// TIA Portal project "XC221_TRABALHOSO" (V12)

(* hardware
DEVICE "S7-1200 station_1"  SIMATIC 1200-Station
   slot 0: "S7-1200 rack"  Rack  V1.0
   slot 1: "PLC_123"  CPU 1214C DC/DC/DC  6ES7 214-1AG31-0XB0  V3.0
   slot 3: "AQ1 x 12 bits"  6ES7 232-4HA30-0XB0  V1.0
*)

// ===== PLC "PLC_123"  CPU 1214C DC/DC/DC =====
// protected blocks, not shown: "EASYPI", "MEMRST"

VAR_GLOBAL   // PLC tag table "Default tag table"
   "System_Byte" AT %MB1 : Byte;
   "FirstScan" AT %M1.0 : Bool;
   "DiagStatusUpdate" AT %M1.1 : Bool;
   "AlwaysTRUE" AT %M1.2 : Bool;
   "AlwaysFALSE" AT %M1.3 : Bool;
   "Clock_Byte" AT %MB0 : Byte;
   "Clock_10Hz" AT %M0.0 : Bool;
   "Clock_5Hz" AT %M0.1 : Bool;
   "Clock_2.5Hz" AT %M0.2 : Bool;
   "Clock_2Hz" AT %M0.3 : Bool;
   "Clock_1.25Hz" AT %M0.4 : Bool;
   "Clock_1Hz" AT %M0.5 : Bool;
   "Clock_0.625Hz" AT %M0.6 : Bool;
   "Clock_0.5Hz" AT %M0.7 : Bool;
   "Tag_1" AT %M31.0 : Bool;
   "Comando_ventilador1" AT %M31.1 : Bool;   // Variavel Auxliar usado no Ventilado 1
   "Comando_ventilador2" AT %M31.2 : Bool;   // Variavel Auxliar usado no Ventilado 2
   "Tag_2" AT %MD701 : Real;
   "Tag_3" AT %MD573 : Real;
   "Tag_4" AT %M203.2 : Bool;
   "Comando_ventilador3" AT %M203.3 : Bool;   // Variavel Auxliar usado no Ventilado 3
   "Comando_ventilador4" AT %M203.4 : Bool;   // Variavel Auxliar usado no Ventilado 4
END_VAR

VAR_GLOBAL   // PLC tag table "11 - Parâmetros"
   "Par_VT101_HorLim" AT %MD705 : Real;   // Limite de Horas do Ventilador 1
   "Par_VT102_HorLim" AT %MD709 : Real;   // Limite de Horas do Ventilador 2
   "Par_LT101_LimHH" AT %MD713 : Real;   // Limite para a condição “Muito Alto” [mm]
   "Par_LT101_LimH" AT %MD717 : Real;   // Limite para a condição “Alto” [mm]
   "Par_LT101_LimL" AT %MD721 : Real;   // Limite para a condição “Baixo" [mm]
   "Par_LT101_LimLL" AT %MD725 : Real;   // Limite para a condição “Muito Baixo” [mm]
   "Par_LT101_LimDsg" AT %MD729 : Real;   // Limite para desligar a bomba[mm]
   "Par_LT101_LimLig" AT %MD733 : Real;   // Limite para ligar a bomba [mm]
   "Par_LC102_SetPoint" AT %MD737 : Real;   // Setpoint [mm]
   "Par_LC102_Prop" AT %MD741 : Real;   // Ganho proporcional
   "Par_LC102_Integ" AT %MD745 : Real;   // Ganho integral [segundos]
   "Par_BA101_HorLim" AT %MD753 : Real;   // Limite de horas da bomba
   "Par_BA101_RefVel" AT %MD757 : Real;   // Referência de velocidade da bomba [%]
END_VAR

VAR_GLOBAL   // PLC tag table "01 - Entradas Digitais"
   "DIn_Geral_Emerge" AT %I0.0 : Bool;   // Ativa condição de emergencia
   "DIn_Geral_Rearma" AT %I0.1 : Bool;   // Rearma defeitos
   "DIn_Geral_SelLoc" AT %I0.2 : Bool;   // Seleciona local (valvula e ventiladores)
   "DIn_VS101_Abre" AT %I0.3 : Bool;   // Botão abre valvula
   "DIn_VS101_Fecha" AT %I0.4 : Bool;   // Botao fecha valvula
   "DIn_VT101_LigDsg" AT %I0.5 : Bool;   // Botão liga/desliga ventilador 1
   "DIn_VT102_LigDsl" AT %I0.6 : Bool;   // Botão liga/desliga ventilador 2
   "DIn_BA101_DisjOff" AT %I0.7 : Bool;   // Disjuntor da bomba desarmado
END_VAR

VAR_GLOBAL   // PLC tag table "02 - Saidas Digitais"
   "Dou_VS101_Abre" AT %Q0.0 : Bool;   // Abre valvula (energiza)
   "Dou_VT101_Liga" AT %Q0.1 : Bool;   // Liga ventilador 1 (energiza)
   "DOu_VT102_Liga" AT %Q0.2 : Bool;   // Liga ventilador 2 (energiza)
END_VAR

VAR_GLOBAL   // PLC tag table "03 - Entradas Analogicas"
   "AIn_LT101_Nivel" AT %IW64 : UInt;   // Nivel de água no tanque [bruto]
END_VAR

VAR_GLOBAL   // PLC tag table "04 - Saidas Analogicas"
   "AOu_BA101_VelBmb" AT %QW64 : UInt;   // Velocidade da bomba [bruto]
END_VAR

VAR_GLOBAL   // PLC tag table "05 - Comando"
   "Cmd_GERAL_Rearma" AT %M101.0 : Bool;   // Rearma defeitos
   "Cmd_VS101_Abre" AT %M102.0 : Bool;   // Abre valvula
   "Cmd_VS101_Fecha" AT %M102.1 : Bool;   // Fecha valvula
   "Cmd_VT101_Liga" AT %M103.0 : Bool;   // Liga ventilador 1
   "Cmd_VT101_Deslig" AT %M103.1 : Bool;   // Desliga ventilador 1
   "Cmd_VT101_HorRst" AT %M103.2 : Bool;   // Zera horimetro ventilador 1
   "Cmd_VT102_Liga" AT %M104.0 : Bool;   // Liga ventilador 2
   "Cmd_VT102_Deslig" AT %M104.1 : Bool;   // Desliga ventilador 2
   "Cmd_VT102_HorRst" AT %M104.2 : Bool;   // Zera horimetro do ventilador 2
   "Cmd_BA101_Liga" AT %M108.0 : Bool;   // Liga bomba
   "Cmd_BA101_Deslig" AT %M108.1 : Bool;   // Desliga bomba
   "Cmd_BA101_HorRst" AT %M108.2 : Bool;   // Zera horimetro da bomba
   "Cmd_BA101_SelMan" AT %M108.3 : Bool;   // Seleciona modo manual da bomba
   "Cmd_BA101_SelAut" AT %M108.4 : Bool;   // Seleciona modo automatico da bomba
   "Cmd_BA101_SelPID" AT %M108.5 : Bool;   // Seleciona modo PID da bomba
   "Cmd_BA101_SelOnOff" AT %M108.6 : Bool;   // Seleciona modo On/Off da bomba
END_VAR

VAR_GLOBAL   // PLC tag table "06 - Estados"
   "STT_geral_LocSel" AT %M201.0 : Bool;   // Local selecionado(Válvula e ventiladores)
   "STT_VS101_Aberta" AT %M202.0 : Bool;   // Válvula aberta(energizada)
   "STT_VT101_Ligado" AT %M203.0 : Bool;   // Ventilador 1 ligado
   "STT_VT101_Defeito" AT %M203.1 : Bool;   // Ventilador 1 com defeito
   "STT_VT102_Ligado" AT %M204.0 : Bool;   // Ventilador 2 ligado
   "STT_VT102_Defeito" AT %M204.1 : Bool;   // Ventilador 2 com defeito
   "STT_LC101_LigBmb" AT %M206.0 : Bool;   // Solicitação do controlador ON/OFF para ligar a bomba
   "STT_BA101_Ligada" AT %M208.0 : Bool;   // Bomba ligada
   "STT_BA101_Defeito" AT %M208.1 : Bool;   // Bomba com defeito
   "STT_BA101_Bloq" AT %M208.2 : Bool;   // Bomba bloqueada
   "STT_BA101_Mansel" AT %M208.3 : Bool;   // Bomba em modo manual
   "STT_BA101_PIDsel" AT %M208.4 : Bool;   // Bomba em modo PID
END_VAR

VAR_GLOBAL   // PLC tag table "07 - Alarmes"
   "Alr_Geral_emerge" AT %M301.0 : Bool;   // Condição de emergencia ativada
   "Alr_VT101_Horfim" AT %M303.0 : Bool;   // Ventilador 1 com horas esgotadas
   "Alr_VT102_Horfim" AT %M304.0 : Bool;   // Ventilador 2 com horas esgotadas
   "Alr_LT101_ExcedHH" AT %M305.0 : Bool;   // Limite "Muito alto" excedido
   "Alr_LT101_ExcedH" AT %M305.1 : Bool;   // limite "alto" excedido
   "Alr_LT101_ExcedL" AT %M305.2 : Bool;   // limite "baixo" excedido
   "Alr_LT101_ExcedLL" AT %M305.3 : Bool;   // limite "muito baixo" excedido
   "Alr_BA101_HorFim" AT %M308.0 : Bool;   // Bomba com horas esgotadas
   "Alr_BA101_DisjOff" AT %M308.1 : Bool;   // Disjuntor da bomba desarmado
END_VAR

VAR_GLOBAL   // PLC tag table "08 - Auxiliares Digitais"
   "DAu_GERAL_Rearma" AT %M401.0 : Bool;   // Algum botão de rearme atuado
   "DAu_GERAL_pul1s0" AT %M401.1 : Bool;   // Pulso de 1 scan a cada 1 segundo
   "DAu_VS101_AbrLoc" AT %M402.0 : Bool;   // Abre via modo local
   "DAu_VS101_AbrRem" AT %M402.1 : Bool;   // Abre via modo remoto
   "DAu_VT101_LigLoc" AT %M403.0 : Bool;   // Liga via modo local
   "DAu_VT101_LigRem" AT %M403.1 : Bool;   // Liga via modo remoto
   "DAu_VT101_EdgLig" AT %M403.2 : Bool;   // Borda para ligar ventilador 1
   "DAu_VT101_EdgDsg" AT %M403.3 : Bool;   // Borda para desligar ventilador 1
   "DAu_VT102_LigLoc" AT %M404.0 : Bool;   // Liga via modo local
   "DAu_VT102_LigRem" AT %M404.1 : Bool;   // Liga via modo remoto
   "DAu_VT102_EdgLig" AT %M404.2 : Bool;   // borda para ligar ventilador 2
   "DAu_VT102_EdgDsg" AT %M404.3 : Bool;   // borda para desligar ventilador 2
   "DAu_BA101_LigMan" AT %M408.0 : Bool;   // liga via modo manual
   "DAu_BA101_LigOnOff" AT %M408.1 : Bool;   // Liga via modo ON/Off
   "DAu_BA101_LigPID" AT %M408.2 : Bool;   // Liga via modo PID
END_VAR

VAR_GLOBAL   // PLC tag table "09 - Auxiliares analógicos"
   "AAu_VT101_Horas" AT %MD505 : Real;   // Horas Trabalhadas do ventilador 1
   "AAu_VT101_Minutos" AT %MD509 : Real;   // Minutos trabalhados do ventilador 1
   "AAu_VT101_Segs" AT %MD513 : Real;   // Segundos trabalhados do ventilador 1
   "AAu_VT102_Horas" AT %MD517 : Real;   // Horas Trabalhadas do ventilador 2
   "AAu_VT102_Minutos" AT %MD521 : Real;   // Minutos trabalhados do ventilador 2
   "AAu_VT102_Segs" AT %MD525 : Real;   // Segundos trabalhados do ventilador 2
   "AAu_LT101_NivelFP" AT %MD533 : Real;   // Nível em formato real [bruto]
   "AAu_LC102_LstErr" AT %MD553 : Real;   // Ùtimo valor de erro
   "AAu_LC102_LstInt" AT %MD557 : Real;   // Último valor da ação intergral
   "AAu_BA101_Horas" AT %MD537 : Real;   // Horas Trabalhadas da bomba
   "AAu_BA101_Minutos" AT %MD541 : Real;   // Minutos trabalhados da bomba
   "AAu_BA101_Segs" AT %MD545 : Real;   // Segundos trabalhados da bomba
   "AAu_BA101_VelBmb" AT %MD549 : Real;   // Velocidade em formato real[bruto]
END_VAR

VAR_GLOBAL   // PLC tag table "10 - Analógicas"
   "Ana_GERAL_AtvCPU" AT %MD601 : Real;   // Sinalizador de atividades da CPU
   "Ana_VT101_HorDec" AT %MD605 : Real;   // Horas restantes do ventilador 1
   "Ana_VT102_HorDec" AT %MD609 : Real;   // Horas restantes do ventilador 2
   "Ana_LT101_Nivel" AT %MD613 : Real;   // Nivel de água no tanque [mm]
   "Ana_LC102_SinCtrl" AT %MD617 : Real;   // Sinal de controle [%]
   "Ana_BA101_HorDec" AT %MD621 : Real;   // Horas restantes da bomba
   "Ana_BA101_VelBmb" AT %MD625 : Real;   // Velocidade atual da bomba [%]
END_VAR

DATA_BLOCK "AUXPRG"   // DB1
TITLE = Variáveis auxiliares para programação
{ S7_Optimized_Access := 'FALSE' }
AUTHOR : Dimitri
VERSION : 0.1
// Posições de memória para uso em temporizadores, contadores, instruções de detecção de borda etc.
   VAR
      "Timer" : Array [1 .. 20] of IEC_TIMER;
      "Counter" : Array [1 .. 20] of IEC_COUNTER;
      Edge : Array [1 .. 20] of Bool;
   END_VAR
BEGIN
END_DATA_BLOCK

DATA_BLOCK "HORIM_DB_VT2"   // DB5
{ S7_Optimized_Access := 'FALSE' }
VERSION : 0.1
// stored: InstanceOfName HORIM_D
"HORIM_D"
BEGIN
END_DATA_BLOCK

DATA_BLOCK "HORIM_DB_VT1"   // DB6
{ S7_Optimized_Access := 'FALSE' }
VERSION : 0.1
// stored: InstanceOfName HORIM_D
"HORIM_D"
BEGIN
END_DATA_BLOCK

// folder: System blocks/Program resources

DATA_BLOCK "IEC_Timer_0_DB"   // DB2
{ S7_Optimized_Access := 'FALSE' }
AUTHOR : Simatic
FAMILY : IEC
NAME : IEC_TMR
VERSION : 1.0
// stored: InstanceOfName ?
"?"
BEGIN
END_DATA_BLOCK

DATA_BLOCK "IEC_Counter_0_DB"   // DB3
{ S7_Optimized_Access := 'FALSE' }
AUTHOR : Simatic
FAMILY : IEC
NAME : CNTR
VERSION : 1.0
// stored: InstanceOfName ?
"?"
BEGIN
END_DATA_BLOCK

DATA_BLOCK "IEC_Timer_0_DB_4"   // DB4
{ S7_Optimized_Access := 'FALSE' }
AUTHOR : Simatic
FAMILY : IEC
NAME : IEC_TMR
VERSION : 1.0
// stored: InstanceOfName ?
"?"
BEGIN
END_DATA_BLOCK

DATA_BLOCK "IEC_Timer_0_DB_5"   // DB7
{ S7_Optimized_Access := 'FALSE' }
AUTHOR : Simatic
FAMILY : IEC
NAME : IEC_TMR
VERSION : 1.0
// stored: InstanceOfName ?
"?"
BEGIN
END_DATA_BLOCK

DATA_BLOCK "IEC_Timer_0_DB_1"   // DB8
{ S7_Optimized_Access := 'FALSE' }
AUTHOR : Simatic
FAMILY : IEC
NAME : IEC_TMR
VERSION : 1.0
// stored: InstanceOfName ?
"?"
BEGIN
END_DATA_BLOCK

DATA_BLOCK "IEC_Timer_0_DB_2"   // DB9
{ S7_Optimized_Access := 'FALSE' }
AUTHOR : Simatic
FAMILY : IEC
NAME : IEC_TMR
VERSION : 1.0
// stored: InstanceOfName ?
"?"
BEGIN
END_DATA_BLOCK

DATA_BLOCK "IEC_Timer_0_DB_3"   // DB10
{ S7_Optimized_Access := 'FALSE' }
AUTHOR : Simatic
FAMILY : IEC
NAME : IEC_TMR
VERSION : 1.0
// stored: InstanceOfName ?
"?"
BEGIN
END_DATA_BLOCK

// folder: (top level)

FUNCTION_BLOCK "HORIM_D"   // FB1, LAD
{ S7_Optimized_Access := 'FALSE' }
VERSION : 0.1
   VAR_INPUT
      clock1s0 : Bool;
      Ligado : Bool;
      Reset : Bool;
      Limite : Real;
   END_VAR
   VAR_OUTPUT
      Restante : Real;
      Alarme : Bool;
   END_VAR
   VAR_IN_OUT
      Segundos : Real;
      Minutos : Real;
      Horas : Real;
   END_VAR
   VAR_TEMP
      AuxSegundos : Bool;
      AuxMinutos : Bool;
      AuxRestante : Real;
   END_VAR
   VAR_TEMP   // added for the SCL form of the ladder/FBD networks
      _w1 : Bool;
   END_VAR
BEGIN

REGION Network 1: SEgundos
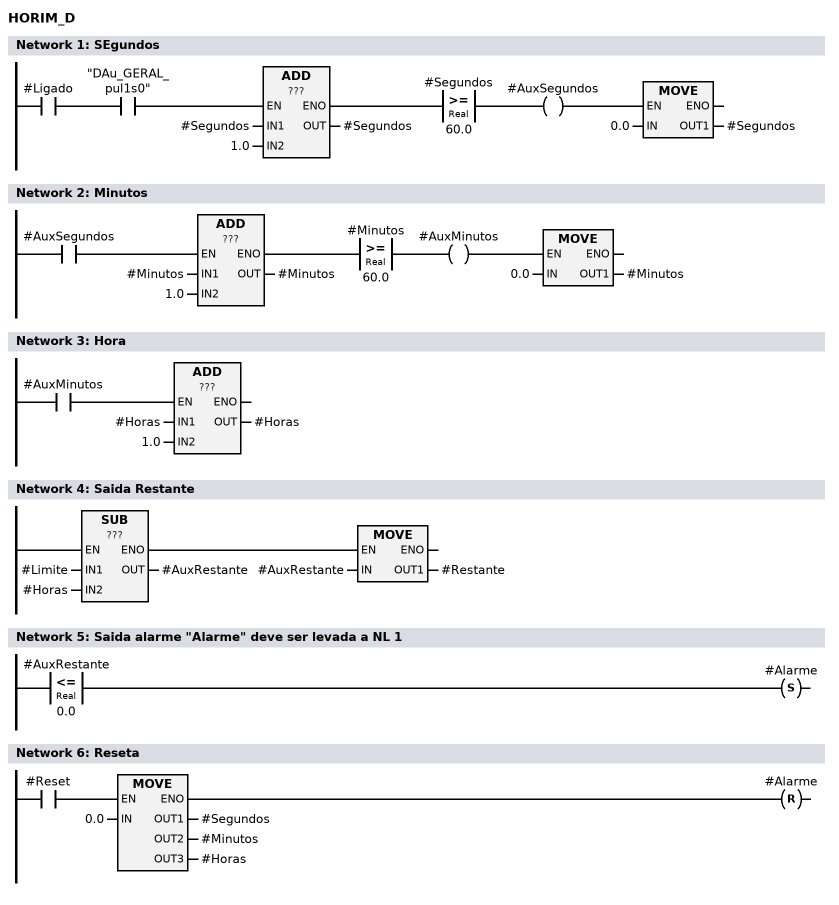
   RUNG wire#powerrail
      Contact( #Ligado )
      Contact( "DAu_GERAL_pul1s0" )
      { S7_Templates := "SrcType := ???"; S7_GenerateENO := "TRUE" } Add(in1 := #Segundos, in2 := 1.0, out => #Segundos)
      { S7_Templates := "SrcType := Real" } GE_Contact(in1 := #Segundos, in2 := 60.0)
      Coil( #AuxSegundos )
      { S7_GenerateENO := "TRUE" } Move(in := 0.0, out1 => #Segundos)
   END_RUNG
   // the same network as SCL:
   // ENO of a box is taken as its EN; it also drops when the box reports an error
   #_w1 := #Ligado AND "DAu_GERAL_pul1s0";
   IF #_w1 THEN #Segundos := #Segundos + 1.0; END_IF;
   #AuxSegundos := #_w1 AND (#Segundos >= 60.0);
   IF #AuxSegundos THEN #Segundos := 0.0; END_IF;
END_REGION

REGION Network 2: Minutos
   RUNG wire#powerrail
      Contact( #AuxSegundos )
      { S7_Templates := "SrcType := ???"; S7_GenerateENO := "TRUE" } Add(in1 := #Minutos, in2 := 1.0, out => #Minutos)
      { S7_Templates := "SrcType := Real" } GE_Contact(in1 := #Minutos, in2 := 60.0)
      Coil( #AuxMinutos )
      { S7_GenerateENO := "TRUE" } Move(in := 0.0, out1 => #Minutos)
   END_RUNG
   // the same network as SCL:
   // ENO of a box is taken as its EN; it also drops when the box reports an error
   IF #AuxSegundos THEN #Minutos := #Minutos + 1.0; END_IF;
   #AuxMinutos := #AuxSegundos AND (#Minutos >= 60.0);
   IF #AuxMinutos THEN #Minutos := 0.0; END_IF;
END_REGION

REGION Network 3: Hora
   RUNG wire#powerrail
      Contact( #AuxMinutos )
      { S7_Templates := "SrcType := ???"; S7_GenerateENO := "TRUE" } Add(in1 := #Horas, in2 := 1.0, out => #Horas)
   END_RUNG
   // the same network as SCL:
   IF #AuxMinutos THEN #Horas := #Horas + 1.0; END_IF;
END_REGION

REGION Network 4: Saida Restante
   RUNG wire#powerrail
      { S7_Templates := "SrcType := ???"; S7_GenerateENO := "TRUE" } Sub(in1 := #Limite, in2 := #Horas, out => #AuxRestante)
      { S7_GenerateENO := "TRUE" } Move(in := #AuxRestante, out1 => #Restante)
   END_RUNG
   // the same network as SCL:
   // ENO of a box is taken as its EN; it also drops when the box reports an error
   #AuxRestante := #Limite - #Horas;
   #Restante := #AuxRestante;
END_REGION

REGION Network 5: Saida alarme "Alarme" deve ser levada a NL 1
   RUNG wire#powerrail
      { S7_Templates := "SrcType := Real" } LE_Contact(in1 := #AuxRestante, in2 := 0.0)
      S_Coil( #Alarme )
   END_RUNG
   // the same network as SCL:
   IF #AuxRestante <= 0.0 THEN #Alarme := TRUE; END_IF;
END_REGION

REGION Network 6: Reseta
   RUNG wire#powerrail
      Contact( #Reset )
      { S7_GenerateENO := "TRUE" } Move(in := 0.0, out1 => #Segundos, out2 => #Minutos, out3 => #Horas)
      R_Coil( #Alarme )
   END_RUNG
   // the same network as SCL:
   // ENO of a box is taken as its EN; it also drops when the box reports an error
   IF #Reset THEN
       #Segundos := 0.0;
       #Minutos := 0.0;
       #Horas := 0.0;
       #Alarme := FALSE;
   END_IF;
END_REGION
END_FUNCTION_BLOCK

FUNCTION "GERAL" : Void   // FC1, LAD
TITLE = Elemento 1 (Elementos Gerais do Sistema):
{ S7_Optimized_Access := 'FALSE' }
VERSION : 0.1
// Bloco que abrange todos os elementos do sistema como o proposito de gerar sinais
BEGIN

REGION Network 1: Condição de emergência ativada (Alarme)
   // É uma váriavel que deve ser levada a nível lógico 1 botão de emergência
   // foi atuado
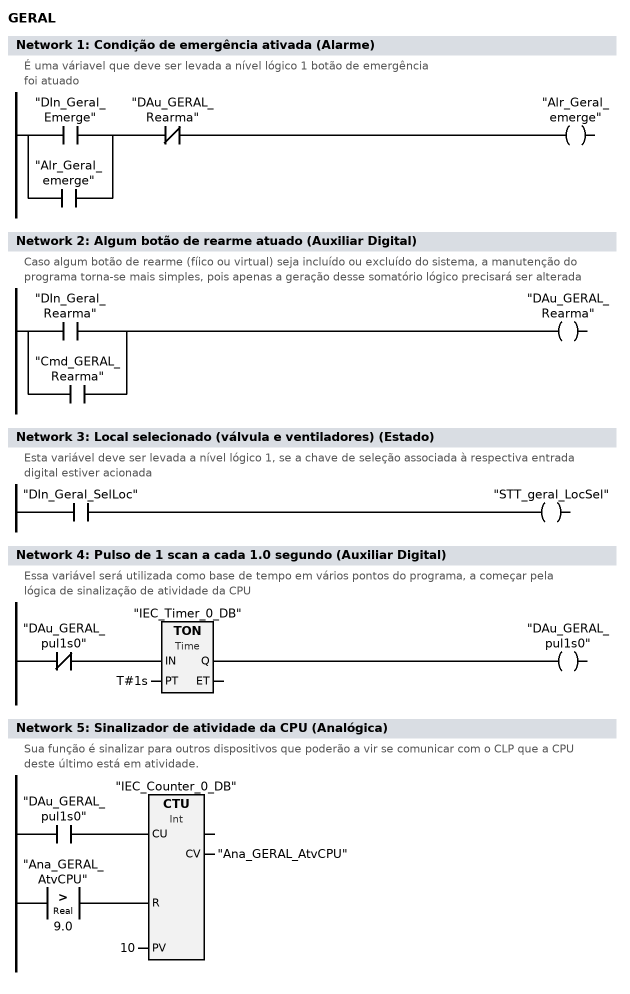
   RUNG wire#powerrail
      Contact( "DIn_Geral_Emerge" )
      wire#w1
      I_Contact( "DAu_GERAL_Rearma" )
      Coil( "Alr_Geral_emerge" )
   END_RUNG
   RUNG wire#powerrail
      Contact( "Alr_Geral_emerge" )
   END_RUNG wire#w1
   // the same network as SCL:
   "Alr_Geral_emerge" := ("DIn_Geral_Emerge" OR "Alr_Geral_emerge") AND NOT "DAu_GERAL_Rearma";
END_REGION

REGION Network 2: Algum botão de rearme atuado (Auxiliar Digital)
   // Caso algum botão de rearme (fíico ou virtual) seja incluído ou excluído do sistema, a manutenção do programa torna-se mais simples, pois apenas a geração desse somatório lógico precisará ser alterada
   RUNG wire#powerrail
      Contact( "DIn_Geral_Rearma" )
      wire#w1
      Coil( "DAu_GERAL_Rearma" )
   END_RUNG
   RUNG wire#powerrail
      Contact( "Cmd_GERAL_Rearma" )
   END_RUNG wire#w1
   // the same network as SCL:
   "DAu_GERAL_Rearma" := "DIn_Geral_Rearma" OR "Cmd_GERAL_Rearma";
END_REGION

REGION Network 3: Local selecionado (válvula e ventiladores) (Estado)
   // Esta variável deve ser levada a nível lógico 1, se a chave de seleção associada à respectiva entrada digital estiver acionada
   RUNG wire#powerrail
      Contact( "DIn_Geral_SelLoc" )
      Coil( "STT_geral_LocSel" )
   END_RUNG
   // the same network as SCL:
   "STT_geral_LocSel" := "DIn_Geral_SelLoc";
END_REGION

REGION Network 4: Pulso de 1 scan a cada 1.0 segundo (Auxiliar Digital)
   // Essa variável será utilizada como base de tempo em vários pontos do programa, a começar pela
   // lógica de sinalização de atividade da CPU
   "IEC_Timer_0_DB".TON(IN := NOT "DAu_GERAL_pul1s0", PT := T#1s);
   "DAu_GERAL_pul1s0" := "IEC_Timer_0_DB".Q;
END_REGION

REGION Network 5: Sinalizador de atividade da CPU (Analógica)
   // Sua função é sinalizar para outros dispositivos que poderão a vir se comunicar com o CLP que a CPU deste último está em atividade.
   "IEC_Counter_0_DB".CTU(CU := "DAu_GERAL_pul1s0",
                          R := "Ana_GERAL_AtvCPU" > 9.0,
                          PV := 10,
                          CV => "Ana_GERAL_AtvCPU");
END_REGION
END_FUNCTION

FUNCTION "VS101" : Void   // FC2, LAD
TITLE = Elemento 2 (Válvula Solenóide):
{ S7_Optimized_Access := 'FALSE' }
VERSION : 0.1
// Este equipamento tem a função de controlar o fluxo de água entre os reservatórios superior e inferior.
BEGIN

REGION Network 1: Abre via modo local (Auxiliar Digital)
   // Abre a valvula solenoide em modo local
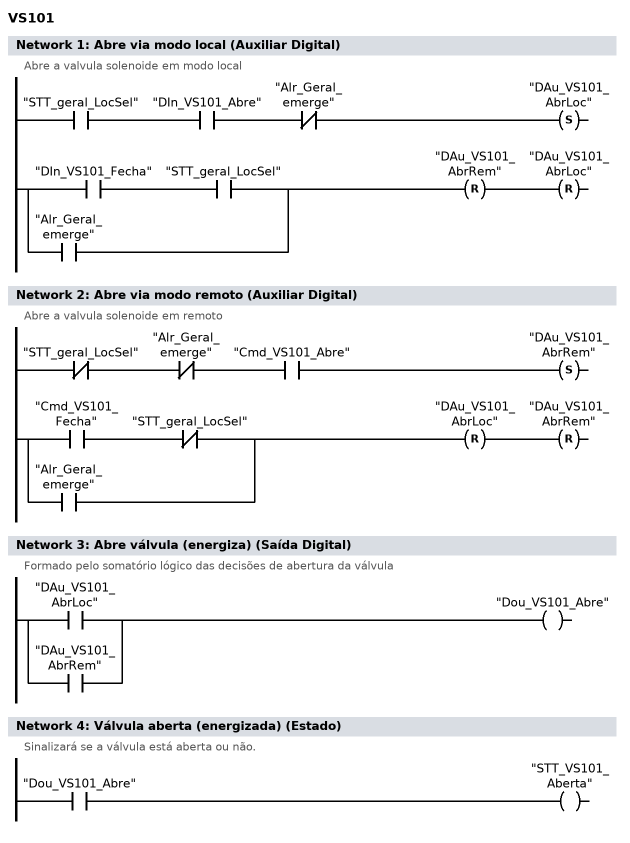
   RUNG wire#powerrail
      Contact( "STT_geral_LocSel" )
      Contact( "DIn_VS101_Abre" )
      I_Contact( "Alr_Geral_emerge" )
      S_Coil( "DAu_VS101_AbrLoc" )
   END_RUNG
   RUNG wire#powerrail
      Contact( "DIn_VS101_Fecha" )
      Contact( "STT_geral_LocSel" )
      wire#w1
      R_Coil( "DAu_VS101_AbrRem" )
      R_Coil( "DAu_VS101_AbrLoc" )
   END_RUNG
   RUNG wire#powerrail
      Contact( "Alr_Geral_emerge" )
   END_RUNG wire#w1
   // the same network as SCL:
   IF "STT_geral_LocSel" AND "DIn_VS101_Abre" AND NOT "Alr_Geral_emerge" THEN
       "DAu_VS101_AbrLoc" := TRUE;
   END_IF;
   IF ("DIn_VS101_Fecha" AND "STT_geral_LocSel") OR "Alr_Geral_emerge" THEN
       "DAu_VS101_AbrRem" := FALSE;
       "DAu_VS101_AbrLoc" := FALSE;
   END_IF;
END_REGION

REGION Network 2: Abre via modo remoto (Auxiliar Digital)
   // Abre a valvula solenoide em remoto
   RUNG wire#powerrail
      I_Contact( "STT_geral_LocSel" )
      I_Contact( "Alr_Geral_emerge" )
      Contact( "Cmd_VS101_Abre" )
      S_Coil( "DAu_VS101_AbrRem" )
   END_RUNG
   RUNG wire#powerrail
      Contact( "Cmd_VS101_Fecha" )
      I_Contact( "STT_geral_LocSel" )
      wire#w1
      R_Coil( "DAu_VS101_AbrLoc" )
      R_Coil( "DAu_VS101_AbrRem" )
   END_RUNG
   RUNG wire#powerrail
      Contact( "Alr_Geral_emerge" )
   END_RUNG wire#w1
   // the same network as SCL:
   IF NOT "STT_geral_LocSel" AND NOT "Alr_Geral_emerge" AND "Cmd_VS101_Abre" THEN
       "DAu_VS101_AbrRem" := TRUE;
   END_IF;
   IF ("Cmd_VS101_Fecha" AND NOT "STT_geral_LocSel") OR "Alr_Geral_emerge" THEN
       "DAu_VS101_AbrLoc" := FALSE;
       "DAu_VS101_AbrRem" := FALSE;
   END_IF;
END_REGION

REGION Network 3: Abre válvula (energiza) (Saída Digital)
   // Formado pelo somatório lógico das decisões de abertura da válvula
   RUNG wire#powerrail
      Contact( "DAu_VS101_AbrLoc" )
      wire#w1
      Coil( "Dou_VS101_Abre" )
   END_RUNG
   RUNG wire#powerrail
      Contact( "DAu_VS101_AbrRem" )
   END_RUNG wire#w1
   // the same network as SCL:
   "Dou_VS101_Abre" := "DAu_VS101_AbrLoc" OR "DAu_VS101_AbrRem";
END_REGION

REGION Network 4: Válvula aberta (energizada) (Estado)
   // Sinalizará se a válvula está aberta ou não.
   RUNG wire#powerrail
      Contact( "Dou_VS101_Abre" )
      Coil( "STT_VS101_Aberta" )
   END_RUNG
   // the same network as SCL:
   "STT_VS101_Aberta" := "Dou_VS101_Abre";
END_REGION
END_FUNCTION

FUNCTION "VT101" : Void   // FC3, LAD
TITLE = Elemento 3 (Ventilador 1)
{ S7_Optimized_Access := 'FALSE' }
VERSION : 0.1
// Bloco para funcionamento do Ventilador 1, porem esse equipamento não está instalado na planta.  Sendo apenas um exemplo hipotetico do que dá pra instalar no projeto. Por isso que o Supervisorio tem que ser de fácil upgrade, a cada novo objeto instalado no ponto equivale a um objeto novo na tela.
BEGIN
END_FUNCTION

FUNCTION "LT101" : Void   // FC4, LAD
TITLE = Elemento 5 (Nível de Água no Tanque)
{ S7_Optimized_Access := 'FALSE' }
VERSION : 0.1
// Nível de água no tanque [mm] (Analógica) . Tem a função de medir o nível de água no reservatório superior.
BEGIN

REGION Network 1: Conversor do valor bruto para tensão
   // A função converte o valor Bruto para real para ser usado na função converte valores
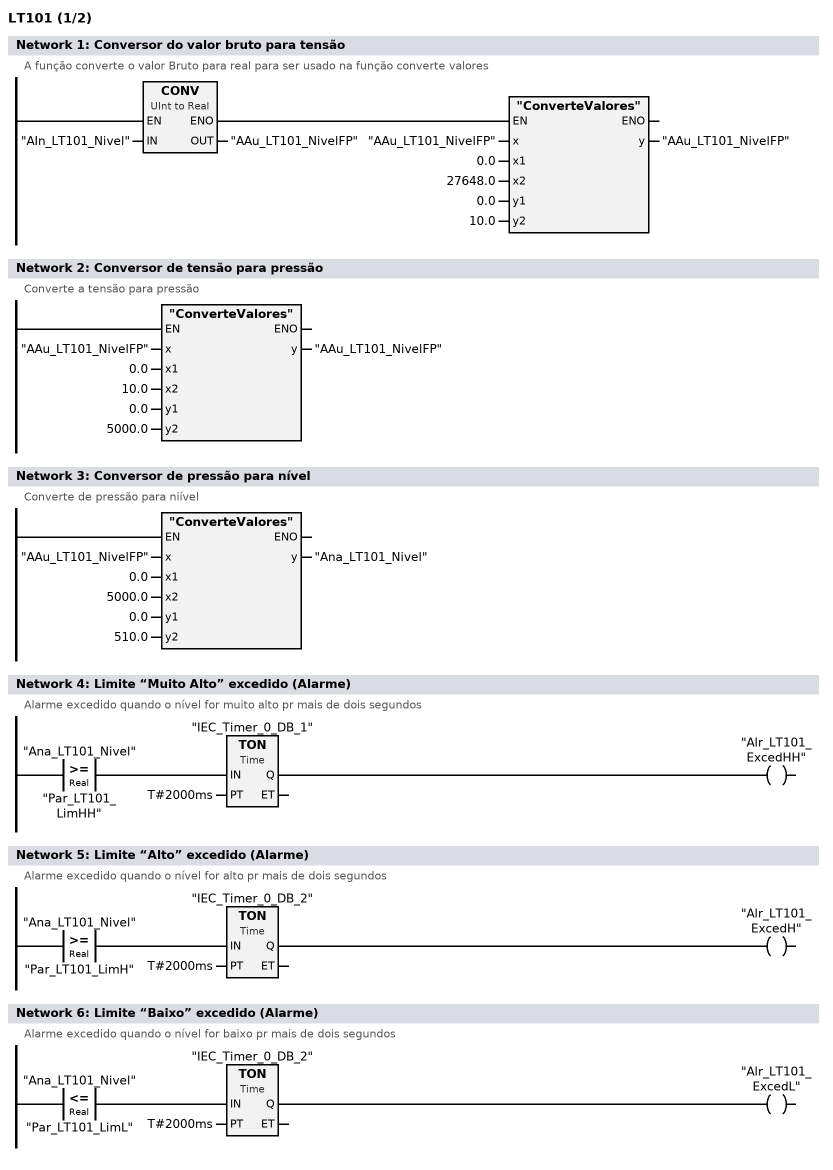
   RUNG wire#powerrail
      { S7_Templates := "[SrcType := UInt, DestType := Real]"; S7_GenerateENO := "TRUE" } Convert(in := "AIn_LT101_Nivel", out => "AAu_LT101_NivelFP")
      "ConverteValores"(x := "AAu_LT101_NivelFP", x1 := 0.0, x2 := 27648.0, y1 := 0.0, y2 := 10.0, y => "AAu_LT101_NivelFP")
   END_RUNG
   // the same network as SCL:
   // ENO of a box is taken as its EN; it also drops when the box reports an error
   "AAu_LT101_NivelFP" := UINT_TO_REAL("AIn_LT101_Nivel");
   "ConverteValores"(x := "AAu_LT101_NivelFP",
                     x1 := 0.0,
                     x2 := 27648.0,
                     y1 := 0.0,
                     y2 := 10.0,
                     y => "AAu_LT101_NivelFP");
END_REGION

REGION Network 2: Conversor de tensão para pressão
   // Converte a tensão para pressão
   RUNG wire#powerrail
      "ConverteValores"(x := "AAu_LT101_NivelFP", x1 := 0.0, x2 := 10.0, y1 := 0.0, y2 := 5000.0, y => "AAu_LT101_NivelFP")
   END_RUNG
   // the same network as SCL:
   "ConverteValores"(x := "AAu_LT101_NivelFP",
                     x1 := 0.0,
                     x2 := 10.0,
                     y1 := 0.0,
                     y2 := 5000.0,
                     y => "AAu_LT101_NivelFP");
END_REGION

REGION Network 3: Conversor de pressão para nível
   // Converte de pressão para niível
   RUNG wire#powerrail
      "ConverteValores"(x := "AAu_LT101_NivelFP", x1 := 0.0, x2 := 5000.0, y1 := 0.0, y2 := 510.0, y => "Ana_LT101_Nivel")
   END_RUNG
   // the same network as SCL:
   "ConverteValores"(x := "AAu_LT101_NivelFP",
                     x1 := 0.0,
                     x2 := 5000.0,
                     y1 := 0.0,
                     y2 := 510.0,
                     y => "Ana_LT101_Nivel");
END_REGION

REGION Network 4: Limite “Muito Alto” excedido (Alarme)
   // Alarme excedido quando o nível for muito alto pr mais de dois segundos
   "IEC_Timer_0_DB_1".TON(IN := "Ana_LT101_Nivel" >= "Par_LT101_LimHH", PT := T#2000ms);
   "Alr_LT101_ExcedHH" := "IEC_Timer_0_DB_1".Q;
END_REGION

REGION Network 5: Limite “Alto” excedido (Alarme)
   // Alarme excedido quando o nível for alto pr mais de dois segundos
   "IEC_Timer_0_DB_2".TON(IN := "Ana_LT101_Nivel" >= "Par_LT101_LimH", PT := T#2000ms);
   "Alr_LT101_ExcedH" := "IEC_Timer_0_DB_2".Q;
END_REGION

REGION Network 6: Limite “Baixo” excedido (Alarme)
   // Alarme excedido quando o nível for baixo pr mais de dois segundos
   "IEC_Timer_0_DB_2".TON(IN := "Ana_LT101_Nivel" <= "Par_LT101_LimL", PT := T#2000ms);
   "Alr_LT101_ExcedL" := "IEC_Timer_0_DB_2".Q;
END_REGION

REGION Network 7: Alarme: excedeu nivel "Muito baixo"
   // Alarme excedido quando o nível for muito baixo por mais de dois segundos
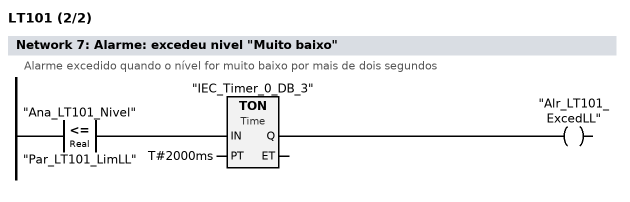
   "IEC_Timer_0_DB_3".TON(IN := "Ana_LT101_Nivel" <= "Par_LT101_LimLL", PT := T#2000ms);
   "Alr_LT101_ExcedLL" := "IEC_Timer_0_DB_3".Q;
END_REGION
END_FUNCTION

FUNCTION "ConverteValores" : Void   // FC5, LAD
{ S7_Optimized_Access := 'FALSE' }
VERSION : 0.1
   VAR_INPUT
      x : Real;
      x1 : Real;
      x2 : Real;
      y1 : Real;
      y2 : Real;
   END_VAR
   VAR_OUTPUT
      y : Real;
   END_VAR
   VAR_TEMP
      "a" : Real;
      "b" : Real;
      Aux1 : Real;
      Aux2 : Real;
   END_VAR
BEGIN

REGION Network 1: Calcular Numerador(Aux 1) e Denomidador (Aux2) do coeficiente angular (#a)
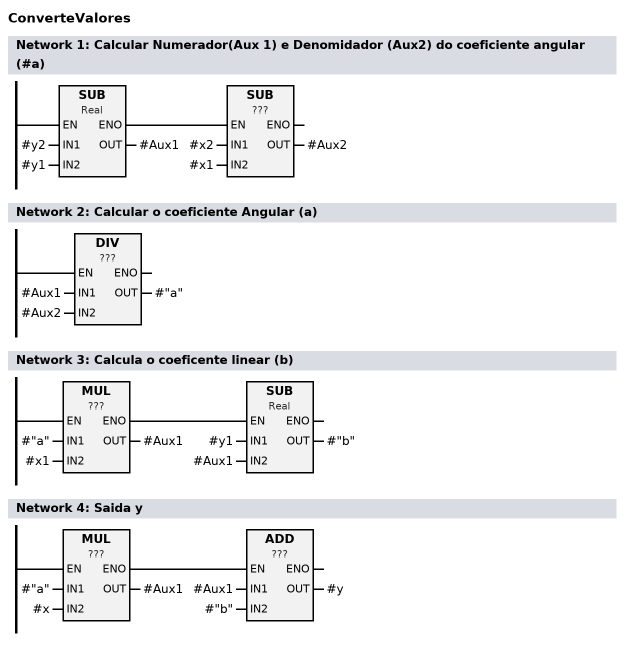
   RUNG wire#powerrail
      { S7_Templates := "SrcType := Real"; S7_GenerateENO := "TRUE" } Sub(in1 := #y2, in2 := #y1, out => #Aux1)
      { S7_Templates := "SrcType := ???"; S7_GenerateENO := "TRUE" } Sub(in1 := #x2, in2 := #x1, out => #Aux2)
   END_RUNG
   // the same network as SCL:
   // ENO of a box is taken as its EN; it also drops when the box reports an error
   #Aux1 := #y2 - #y1;
   #Aux2 := #x2 - #x1;
END_REGION

REGION Network 2: Calcular o coeficiente Angular (a)
   RUNG wire#powerrail
      { S7_Templates := "SrcType := ???"; S7_GenerateENO := "TRUE" } Div(in1 := #Aux1, in2 := #Aux2, out => #"a")
   END_RUNG
   // the same network as SCL:
   #"a" := #Aux1 / #Aux2;
END_REGION

REGION Network 3: Calcula o coeficente linear (b)
   RUNG wire#powerrail
      { S7_Templates := "SrcType := ???"; S7_GenerateENO := "TRUE" } Mul(in1 := #"a", in2 := #x1, out => #Aux1)
      { S7_Templates := "SrcType := Real"; S7_GenerateENO := "TRUE" } Sub(in1 := #y1, in2 := #Aux1, out => #"b")
   END_RUNG
   // the same network as SCL:
   // ENO of a box is taken as its EN; it also drops when the box reports an error
   #Aux1 := #"a" * #x1;
   #"b" := #y1 - #Aux1;
END_REGION

REGION Network 4: Saida y
   RUNG wire#powerrail
      { S7_Templates := "SrcType := ???"; S7_GenerateENO := "TRUE" } Mul(in1 := #"a", in2 := #x, out => #Aux1)
      { S7_Templates := "SrcType := ???"; S7_GenerateENO := "TRUE" } Add(in1 := #Aux1, in2 := #"b", out => #y)
   END_RUNG
   // the same network as SCL:
   // ENO of a box is taken as its EN; it also drops when the box reports an error
   #Aux1 := #"a" * #x;
   #y := #Aux1 + #"b";
END_REGION
END_FUNCTION

FUNCTION "VT102" : Void   // FC6, LAD
TITLE = Elemento 4 (Ventilador 2)
{ S7_Optimized_Access := 'FALSE' }
VERSION : 0.1
// Bloco para funcionamento do Ventilador 1, porem esse equipamento não está instalado na planta.  Sendo apenas um exemplo hipotetico do que dá pra instalar no projeto. Por isso que o Supervisorio tem que ser de fácil upgrade, a cada novo objeto instalado no ponto equivale a um objeto novo na tela.
BEGIN
END_FUNCTION

FUNCTION "HORIM" : Void   // FC7, LAD
{ S7_Optimized_Access := 'FALSE' }
VERSION : 0.1
   VAR_INPUT
      clock1s0 : Bool;
      Ligado : Bool;
      Reset : Bool;
      Limite : Real;
   END_VAR
   VAR_OUTPUT
      Restante : Real;
      Alarme : Bool;
   END_VAR
   VAR_IN_OUT
      Segundos : Real;
      Minutos : Real;
      Horas : Real;
   END_VAR
   VAR_TEMP
      AuxSegundos : Bool;
      AuxMinutos : Bool;
      AuxRestante : Real;
   END_VAR
   VAR_TEMP   // added for the SCL form of the ladder/FBD networks
      _w1 : Bool;
   END_VAR
BEGIN

REGION Network 1: SEgundos
   // Conta ate 60 segundos, incrementa um minuto na network 2, recomeca a contagem a partir de zero.
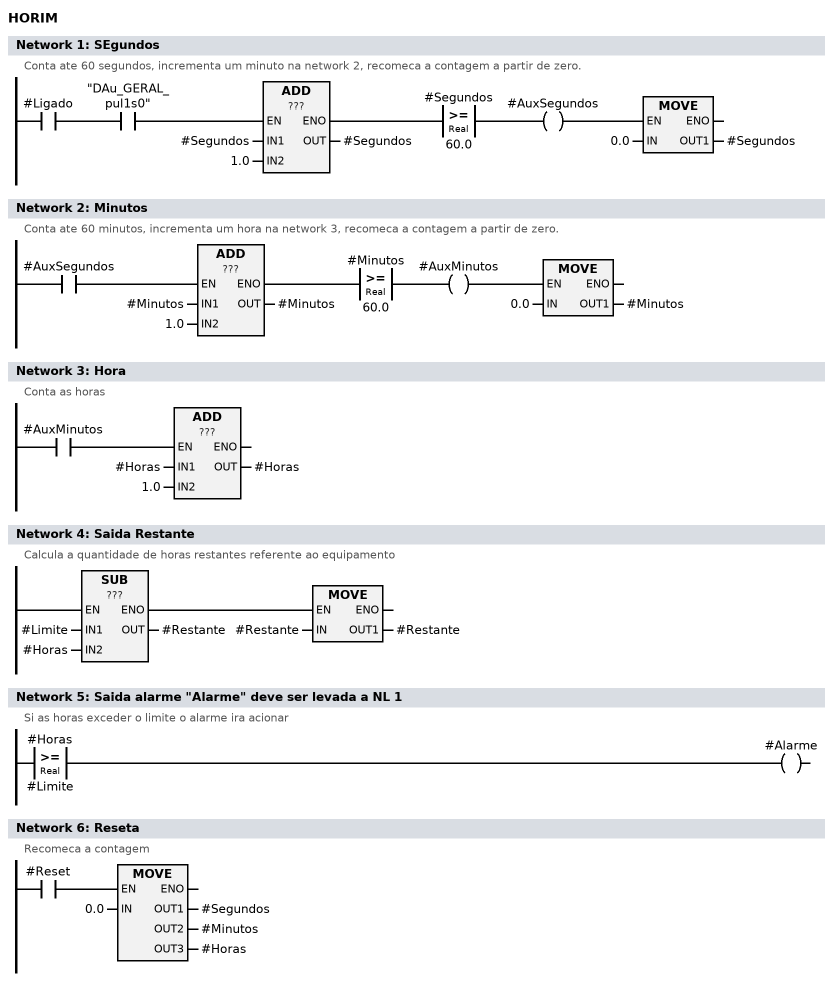
   RUNG wire#powerrail
      Contact( #Ligado )
      Contact( "DAu_GERAL_pul1s0" )
      { S7_Templates := "SrcType := ???"; S7_GenerateENO := "TRUE" } Add(in1 := #Segundos, in2 := 1.0, out => #Segundos)
      { S7_Templates := "SrcType := Real" } GE_Contact(in1 := #Segundos, in2 := 60.0)
      Coil( #AuxSegundos )
      { S7_GenerateENO := "TRUE" } Move(in := 0.0, out1 => #Segundos)
   END_RUNG
   // the same network as SCL:
   // ENO of a box is taken as its EN; it also drops when the box reports an error
   #_w1 := #Ligado AND "DAu_GERAL_pul1s0";
   IF #_w1 THEN #Segundos := #Segundos + 1.0; END_IF;
   #AuxSegundos := #_w1 AND (#Segundos >= 60.0);
   IF #AuxSegundos THEN #Segundos := 0.0; END_IF;
END_REGION

REGION Network 2: Minutos
   // Conta ate 60 minutos, incrementa um hora na network 3, recomeca a contagem a partir de zero.
   RUNG wire#powerrail
      Contact( #AuxSegundos )
      { S7_Templates := "SrcType := ???"; S7_GenerateENO := "TRUE" } Add(in1 := #Minutos, in2 := 1.0, out => #Minutos)
      { S7_Templates := "SrcType := Real" } GE_Contact(in1 := #Minutos, in2 := 60.0)
      Coil( #AuxMinutos )
      { S7_GenerateENO := "TRUE" } Move(in := 0.0, out1 => #Minutos)
   END_RUNG
   // the same network as SCL:
   // ENO of a box is taken as its EN; it also drops when the box reports an error
   IF #AuxSegundos THEN #Minutos := #Minutos + 1.0; END_IF;
   #AuxMinutos := #AuxSegundos AND (#Minutos >= 60.0);
   IF #AuxMinutos THEN #Minutos := 0.0; END_IF;
END_REGION

REGION Network 3: Hora
   // Conta as horas
   RUNG wire#powerrail
      Contact( #AuxMinutos )
      { S7_Templates := "SrcType := ???"; S7_GenerateENO := "TRUE" } Add(in1 := #Horas, in2 := 1.0, out => #Horas)
   END_RUNG
   // the same network as SCL:
   IF #AuxMinutos THEN #Horas := #Horas + 1.0; END_IF;
END_REGION

REGION Network 4: Saida Restante
   // Calcula a quantidade de horas restantes referente ao equipamento
   RUNG wire#powerrail
      { S7_Templates := "SrcType := ???"; S7_GenerateENO := "TRUE" } Sub(in1 := #Limite, in2 := #Horas, out => #Restante)
      { S7_GenerateENO := "TRUE" } Move(in := #Restante, out1 => #Restante)
   END_RUNG
   // the same network as SCL:
   // ENO of a box is taken as its EN; it also drops when the box reports an error
   #Restante := #Limite - #Horas;
   #Restante := #Restante;
END_REGION

REGION Network 5: Saida alarme "Alarme" deve ser levada a NL 1
   // Si as horas exceder o limite o alarme ira acionar
   RUNG wire#powerrail
      { S7_Templates := "SrcType := Real" } GE_Contact(in1 := #Horas, in2 := #Limite)
      Coil( #Alarme )
   END_RUNG
   // the same network as SCL:
   #Alarme := #Horas >= #Limite;
END_REGION

REGION Network 6: Reseta
   // Recomeca a contagem
   RUNG wire#powerrail
      Contact( #Reset )
      { S7_GenerateENO := "TRUE" } Move(in := 0.0, out1 => #Segundos, out2 => #Minutos, out3 => #Horas)
   END_RUNG
   // the same network as SCL:
   IF #Reset THEN
       #Segundos := 0.0;
       #Minutos := 0.0;
       #Horas := 0.0;
   END_IF;
END_REGION
END_FUNCTION

FUNCTION "LC101" : Void   // FC8, LAD
TITLE = Elemento 6 (Controlador On/Off de Nível):
{ S7_Optimized_Access := 'FALSE' }
VERSION : 0.1
// Este controlador tem a função de ligar e desligar a bomba de água de forma que o nível no reservatório superior seja mantido dentro de uma determinada faixa.
BEGIN

REGION Network 1: Solicitação do controlador On/Off para ligar bomba (Estado)
   // Se o nivel de agua no tanque for menor do que o limite para ligar a bomba por mais de 1 segundo então deve se setar a bomba (ligar)
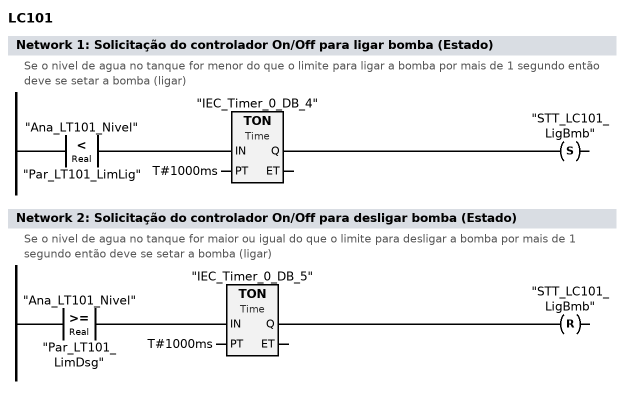
   "IEC_Timer_0_DB_4".TON(IN := "Ana_LT101_Nivel" < "Par_LT101_LimLig", PT := T#1000ms);
   IF "IEC_Timer_0_DB_4".Q THEN "STT_LC101_LigBmb" := TRUE; END_IF;
END_REGION

REGION Network 2: Solicitação do controlador On/Off para desligar bomba (Estado)
   // Se o nivel de agua no tanque for maior ou igual do que o limite para desligar a bomba por mais de 1 segundo então deve se setar a bomba (ligar)
   "IEC_Timer_0_DB_5".TON(IN := "Ana_LT101_Nivel" >= "Par_LT101_LimDsg", PT := T#1000ms);
   IF "IEC_Timer_0_DB_5".Q THEN "STT_LC101_LigBmb" := FALSE; END_IF;
END_REGION
END_FUNCTION

FUNCTION "BA101" : Void   // FC10, LAD
TITLE = Elemento 8 (Bomba deÁgua):
{ S7_Optimized_Access := 'FALSE' }
VERSION : 0.1
// A função desse equipamento é bombear a água do reservatório inferior para o reservatório superior.
BEGIN
END_FUNCTION

ORGANIZATION_BLOCK "Main"   // OB1, LAD, ProgramCycle
TITLE = Ciclo principal do programa
{ S7_Optimized_Access := 'FALSE' }
VERSION : 0.1
   VAR_TEMP   // added for the SCL form of the ladder/FBD networks
      _w1 : Bool;
   END_VAR
BEGIN

REGION Network 1: Geral
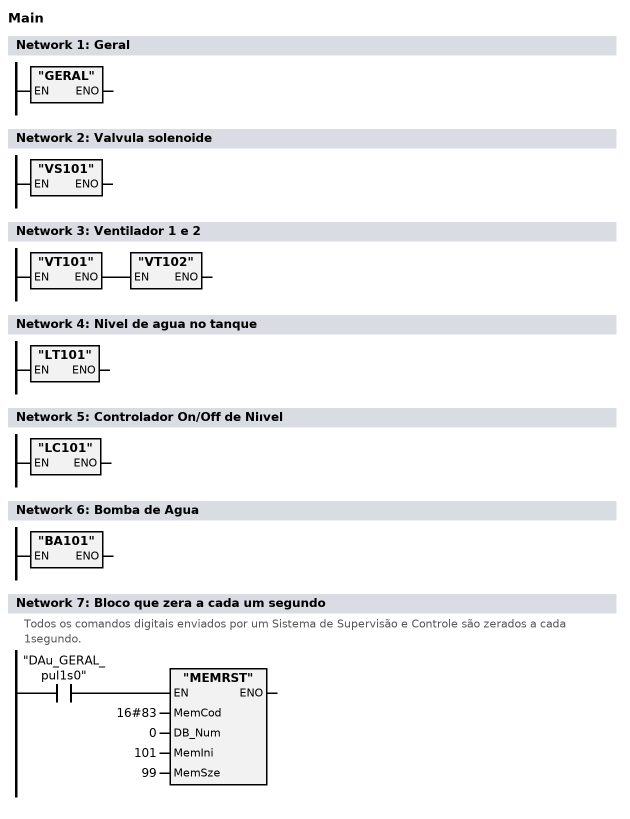
   RUNG wire#powerrail
      "GERAL"()
   END_RUNG
   // the same network as SCL:
   "GERAL"();
END_REGION

REGION Network 2: Valvula solenoide
   RUNG wire#powerrail
      "VS101"()
   END_RUNG
   // the same network as SCL:
   "VS101"();
END_REGION

REGION Network 3: Ventilador 1 e 2
   RUNG wire#powerrail
      "VT101"()
      "VT102"()
   END_RUNG
   // the same network as SCL:
   "VT101"(ENO => #_w1);
   IF #_w1 THEN "VT102"(); END_IF;
END_REGION

REGION Network 4: Nivel de agua no tanque
   RUNG wire#powerrail
      "LT101"()
   END_RUNG
   // the same network as SCL:
   "LT101"();
END_REGION

REGION Network 5: Controlador On/Off de Niıvel
   RUNG wire#powerrail
      "LC101"()
   END_RUNG
   // the same network as SCL:
   "LC101"();
END_REGION

REGION Network 6: Bomba de Agua
   RUNG wire#powerrail
      "BA101"()
   END_RUNG
   // the same network as SCL:
   "BA101"();
END_REGION

REGION Network 7: Bloco que zera a cada um segundo
   // Todos os comandos digitais enviados por um Sistema de Supervisão e Controle são zerados a cada 1segundo.
   RUNG wire#powerrail
      Contact( "DAu_GERAL_pul1s0" )
      "MEMRST"(MemCod := 16#83, DB_Num := 0, MemIni := 101, MemSze := 99)
   END_RUNG
   // the same network as SCL:
   IF "DAu_GERAL_pul1s0" THEN "MEMRST"(MemCod := 16#83, DB_Num := 0, MemIni := 101, MemSze := 99); END_IF;
END_REGION
END_ORGANIZATION_BLOCK

ORGANIZATION_BLOCK "LC102"   // OB30, LAD, CyclicInterrupt
TITLE = Elemento 7 (Controlador PID de Nível)
{ S7_Optimized_Access := 'FALSE' }
VERSION : 0.1
// Este controlador tem a função de determinar a velocidade ideal para a bomba de água de forma a minimizar a diferença entre o valor desejado para o nível do reservatório superior e o valor real dessa grandeza.
BEGIN

REGION Network 1: Chama o bloco do PID e seta as variaveis
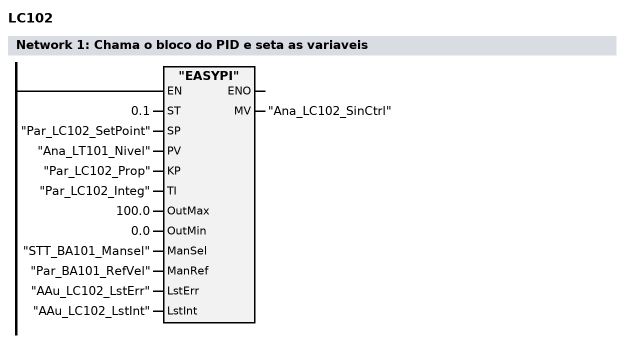
   RUNG wire#powerrail
      "EASYPI"(ST := 0.1, SP := "Par_LC102_SetPoint", PV := "Ana_LT101_Nivel", KP := "Par_LC102_Prop", TI := "Par_LC102_Integ", OutMax := 100.0, OutMin := 0.0, ManSel := "STT_BA101_Mansel", ManRef := "Par_BA101_RefVel", LstErr := "AAu_LC102_LstErr", LstInt := "AAu_LC102_LstInt", MV => "Ana_LC102_SinCtrl")
   END_RUNG
   // the same network as SCL:
   "EASYPI"(ST := 0.1,
            SP := "Par_LC102_SetPoint",
            PV := "Ana_LT101_Nivel",
            KP := "Par_LC102_Prop",
            TI := "Par_LC102_Integ",
            OutMax := 100.0,
            OutMin := 0.0,
            ManSel := "STT_BA101_Mansel",
            ManRef := "Par_BA101_RefVel",
            LstErr := "AAu_LC102_LstErr",
            LstInt := "AAu_LC102_LstInt",
            MV => "Ana_LC102_SinCtrl");
END_REGION
END_ORGANIZATION_BLOCK

ORGANIZATION_BLOCK "Startup"   // OB100, LAD, Startup
TITLE = Bloco Startup
{ S7_Optimized_Access := 'FALSE' }
VERSION : 0.1
   VAR_INPUT
      LostRetentive : Bool;   // True if retentive data are lost
      LostRTC : Bool;   // True if date and time are lost
   END_VAR
BEGIN
END_ORGANIZATION_BLOCK